// TIA Portal V15.1 export
// export: Created 2024-06-21T08:40:52.4379165Z, ExportSetting WithDefaults, DisplayName Totally Integrated Automation Portal, DisplayVersion V15.1 Update 5, DisplayName TIA Portal Openness, DisplayVersion V15.1 Update 5, DisplayName SINAMICS Startdrive Advanced, DisplayVersion V15.1, DisplayName G130, G150, S120, S150, SINAMICS MV, S210, DisplayVersion V15.1, DisplayName G110M, G120, G120C, G120D, G120P, DisplayVersion V15.1, DisplayName STEP 7 Professional, DisplayVersion V15.1 Update 5, DisplayName STEP 7 Safety, DisplayVersion V15.1, DisplayName WinCC Professional, DisplayVersion V15.1 Update 5, DisplayName SIMATIC Visualization Architect, DisplayVersion V15.1
FUNCTION_BLOCK "LTimer"   // FB1009, FBD
TITLE = LTimer
{ S7_Optimized_Access := 'FALSE' }
AUTHOR : VCC
FAMILY : Control
NAME : TimerON
VERSION : 1.0
// ================================================================================
// LTimer is used when a delay is necessary without using a hardware timer.
// The output of the timer will follow the input after a delay time. When the 
// input 
// drops to False, the output will drop immediatly.
// 
// During the activation of timer, hold input can freeze the timer
// * Input Hold = false then normal running of timer
// * Input Hold = true then timer frozen.
// ================================================================================
// stored: AutoNumber false, IsIECCheckEnabled false, SetENOAutomatically False, UDAEnableTagReadback false
   VAR_INPUT
      I_StartTimer { ExternalAccessible := 'False'; ExternalVisible := 'False'; ExternalWritable := 'False'} : Bool;   // Start Timer
      I_HoldTimer { ExternalAccessible := 'False'; ExternalVisible := 'False'; ExternalWritable := 'False'} : Bool;   // Hold timer
      I_MaxTimerValue { ExternalAccessible := 'False'; ExternalVisible := 'False'; ExternalWritable := 'False'} : DInt;   // Maximum Timer Value (1 unit = 1ms and max=7FFFFFFF)
   END_VAR
   VAR_OUTPUT
      O_TimerResult { ExternalAccessible := 'False'; ExternalVisible := 'False'; ExternalWritable := 'False'} : Bool;   // Timer result when time = MaxTime
      O_TimerValue { ExternalAccessible := 'False'; ExternalVisible := 'False'; ExternalWritable := 'False'} : DInt;   // Current timer value
   END_VAR
   VAR DB_SPECIFIC
      PrevCPUSystemTime { ExternalAccessible := 'False'; ExternalVisible := 'False'; ExternalWritable := 'False'} : DInt;   // Last value of the CPU system time register
      DeltaCpuTime { ExternalAccessible := 'False'; ExternalVisible := 'False'; ExternalWritable := 'False'} : DInt;   // Time difference of CPU System Time register compared with last scan
      TempDInt1 { ExternalAccessible := 'False'; ExternalVisible := 'False'; ExternalWritable := 'False'} : DInt;   // Just a temporary Double Integer value
      TimerValue { ExternalAccessible := 'False'; ExternalVisible := 'False'; ExternalWritable := 'False'} : DInt;   // Current timer value
   END_VAR
BEGIN

REGION Network 1: **** 4.4 - Machine Status - Calculated **** Set #TimerValue to zero whenever it a negative.
   // Set #TimerValue to zero whenever it a negative.
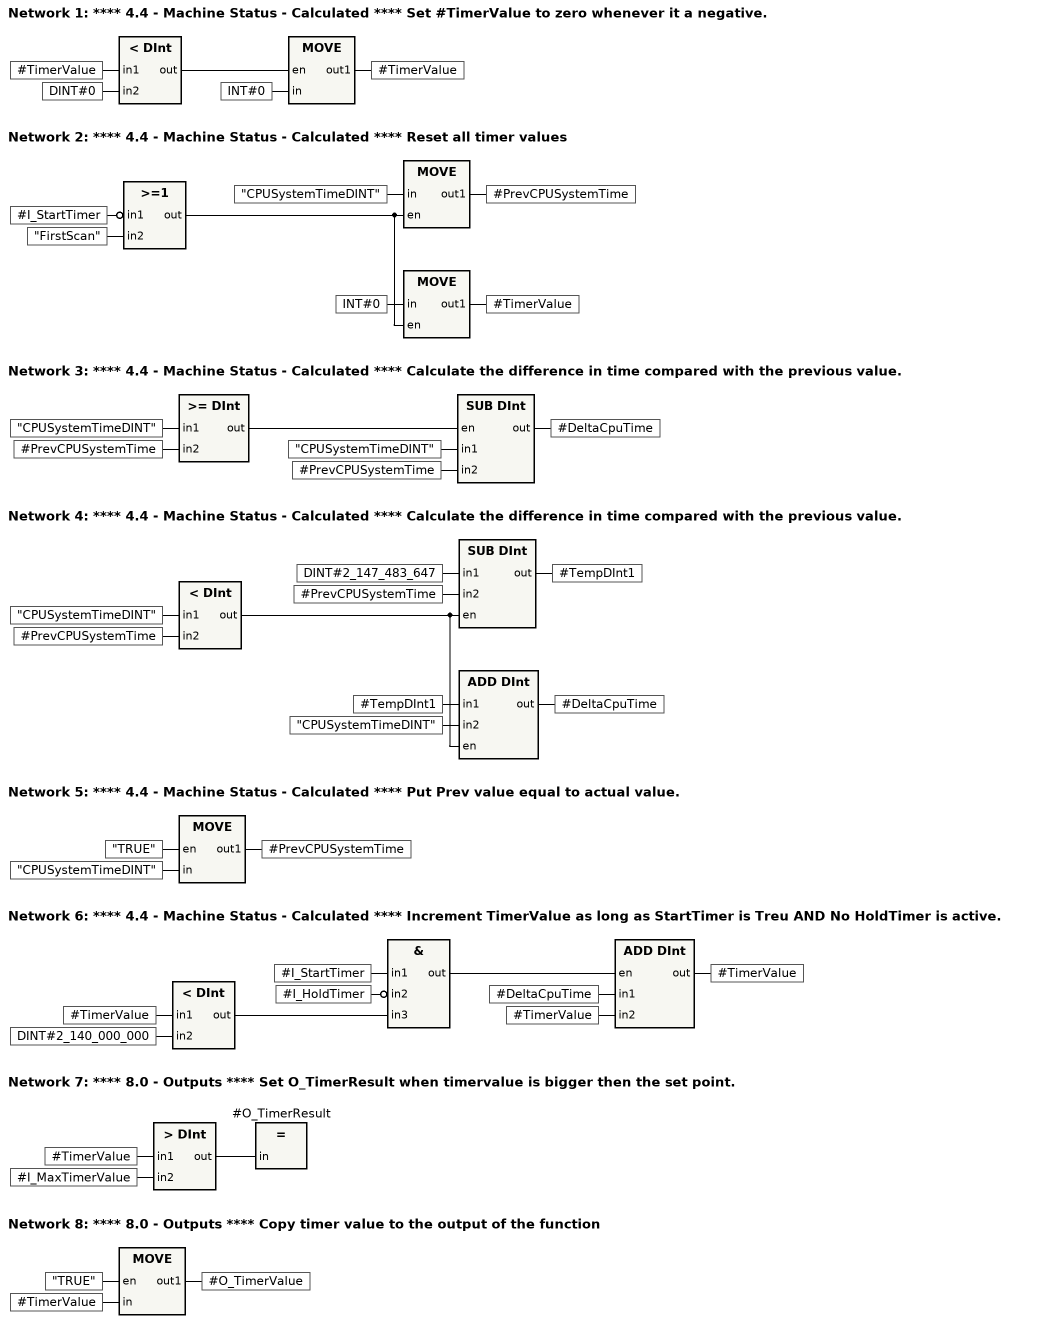
   IF #TimerValue < DINT#0 THEN #TimerValue := INT#0; END_IF;
END_REGION

REGION Network 2: **** 4.4 - Machine Status - Calculated **** Reset all timer values
   // Reset all timer values
   IF NOT #I_StartTimer OR "FirstScan" THEN
       #PrevCPUSystemTime := "CPUSystemTimeDINT";
       #TimerValue := INT#0;
   END_IF;
END_REGION

REGION Network 3: **** 4.4 - Machine Status - Calculated **** Calculate the difference in time compared with the previous value.
   // Calculate the difference in time compared with the previous value.
   IF "CPUSystemTimeDINT" >= #PrevCPUSystemTime THEN
       #DeltaCpuTime := "CPUSystemTimeDINT" - #PrevCPUSystemTime;
   END_IF;
END_REGION

REGION Network 4: **** 4.4 - Machine Status - Calculated **** Calculate the difference in time compared with the previous value.
   // Calculate the difference in time compared with the previous value.
   // If the cpu time has passed 2147483647 then the delta is used first.
   IF "CPUSystemTimeDINT" < #PrevCPUSystemTime THEN
       #TempDInt1 := DINT#2_147_483_647 - #PrevCPUSystemTime;
       #DeltaCpuTime := #TempDInt1 + "CPUSystemTimeDINT";
   END_IF;
END_REGION

REGION Network 5: **** 4.4 - Machine Status - Calculated **** Put Prev value equal to actual value.
   // Put Prev value equal to actual value.
   IF "TRUE" THEN #PrevCPUSystemTime := "CPUSystemTimeDINT"; END_IF;
END_REGION

REGION Network 6: **** 4.4 - Machine Status - Calculated **** Increment TimerValue as long as StartTimer is Treu AND No HoldTimer is active.
   // Increment TimerValue as long as StartTimer is Treu AND No HoldTimer is active.
   // Make sure that there is no override by limiting the increment.
   IF #I_StartTimer AND NOT #I_HoldTimer AND (#TimerValue < DINT#2_140_000_000) THEN
       #TimerValue := #DeltaCpuTime + #TimerValue;
   END_IF;
END_REGION

REGION Network 7: **** 8.0 - Outputs **** Set O_TimerResult when timervalue is bigger then the set point.
   // Set O_TimerResult when timervalue is bigger then the set point.
   #O_TimerResult := #TimerValue > #I_MaxTimerValue;
END_REGION

REGION Network 8: **** 8.0 - Outputs **** Copy timer value to the output of the function
   // Copy timer value to the output of the function
   IF "TRUE" THEN #O_TimerValue := #TimerValue; END_IF;
END_REGION
END_FUNCTION_BLOCK
